Staubli VAL3: language.pjx

--- language.pjx ---
Parameters version=s7.1 stackSize=5000 millimeterUnit=true
Program file=getLanguage.pgx
Program file=getYesNo.pgx
Program file=message.pgx
Program file=page.pgx
Program file=setLanguage.pgx
Data file=language.dtx
Library alias=language path=Disk://kernel/language/english/english.pjx

--- setLanguage.pgx ---
public program setLanguage(string x_sPath)
  local num l_nResult
  local string l_sMessage
begin
  //
  call language:message(l_sMessage,-7)
  l_nResult=language:libLoad(x_sPath)
  delay(0)
  if l_nResult!=0
    popUpMsg(l_sMessage+x_sPath+" ; "+toString("",l_nResult))
  endIf
end
